FUNCTION_BLOCK UA_SkillFacade (* OPC UA object of one skill: one method per PackML command (answered synchronously with Accepted/ErrorID) and published State, ErrorID and latched parameters *)
  (* Standard: 61499-2 *)
  (* Version 2.0, 2026-09-27, Project contributors, Filling cell reference model *)
  PACKAGE fillingcell;
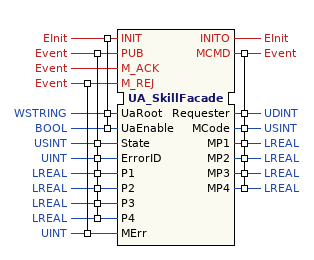
  EVENT_INPUT
    INIT : EInit WITH UaRoot, UaEnable;
    PUB WITH State, ErrorID, P1, P2, P3, P4;
    M_ACK;
    M_REJ WITH MErr;
  END_EVENT
  EVENT_OUTPUT
    INITO : EInit;
    MCMD WITH Requester, MCode, MP1, MP2, MP3, MP4;
  END_EVENT
  VAR_INPUT
    UaRoot : WSTRING;
    UaEnable : BOOL;
    State : USINT;
    ErrorID : UINT;
    P1 : LREAL;
    P2 : LREAL;
    P3 : LREAL;
    P4 : LREAL;
    MErr : UINT;
  END_VAR
  VAR_OUTPUT
    Requester : UDINT;
    MCode : USINT;
    MP1 : LREAL;
    MP2 : LREAL;
    MP3 : LREAL;
    MP4 : LREAL;
  END_VAR
  FBS
    Ids : fillingcell::UA_SkillIds;
    Calls : fillingcell::UA_SkillMux;
    Srv_Reset : iec61499::net::SERVER_2_1;
    Srv_Start : iec61499::net::SERVER_2_5;
    Srv_Hold : iec61499::net::SERVER_2_1;
    Srv_Unhold : iec61499::net::SERVER_2_1;
    Srv_Stop : iec61499::net::SERVER_2_1;
    Srv_Abort : iec61499::net::SERVER_2_1;
    Srv_Clear : iec61499::net::SERVER_2_1;
    Publisher : iec61499::net::PUBLISH_6;
  END_FBS
  EVENT_CONNECTIONS
    Srv_Reset.IND TO Calls.IND_Reset;
    Calls.RSP_Reset TO Srv_Reset.RSP;
    Srv_Start.IND TO Calls.IND_Start;
    Calls.RSP_Start TO Srv_Start.RSP;
    Srv_Hold.IND TO Calls.IND_Hold;
    Calls.RSP_Hold TO Srv_Hold.RSP;
    Srv_Unhold.IND TO Calls.IND_Unhold;
    Calls.RSP_Unhold TO Srv_Unhold.RSP;
    Srv_Stop.IND TO Calls.IND_Stop;
    Calls.RSP_Stop TO Srv_Stop.RSP;
    Srv_Abort.IND TO Calls.IND_Abort;
    Calls.RSP_Abort TO Srv_Abort.RSP;
    Srv_Clear.IND TO Calls.IND_Clear;
    Calls.RSP_Clear TO Srv_Clear.RSP;
    INIT TO Ids.INIT;
    Ids.INITO TO Srv_Reset.INIT;
    Srv_Reset.INITO TO Srv_Start.INIT;
    Srv_Start.INITO TO Srv_Hold.INIT;
    Srv_Hold.INITO TO Srv_Unhold.INIT;
    Srv_Unhold.INITO TO Srv_Stop.INIT;
    Srv_Stop.INITO TO Srv_Abort.INIT;
    Srv_Abort.INITO TO Srv_Clear.INIT;
    Srv_Clear.INITO TO Publisher.INIT;
    Publisher.INITO TO INITO;
    PUB TO Publisher.REQ;
    Calls.S_CMD TO MCMD;
    M_ACK TO Calls.S_ACK;
    M_REJ TO Calls.S_REJ;
  END_CONNECTIONS
  DATA_CONNECTIONS
    UaEnable TO Srv_Reset.QI;
    Ids.Id_Reset TO Srv_Reset.ID;
    Srv_Reset.RD_1 TO Calls.Req_Reset;
    Calls.Accepted TO Srv_Reset.SD_1;
    Calls.ErrorID TO Srv_Reset.SD_2;
    UaEnable TO Srv_Start.QI;
    Ids.Id_Start TO Srv_Start.ID;
    Srv_Start.RD_1 TO Calls.Req_Start;
    Srv_Start.RD_2 TO Calls.Start_P1;
    Srv_Start.RD_3 TO Calls.Start_P2;
    Srv_Start.RD_4 TO Calls.Start_P3;
    Srv_Start.RD_5 TO Calls.Start_P4;
    Calls.Accepted TO Srv_Start.SD_1;
    Calls.ErrorID TO Srv_Start.SD_2;
    UaEnable TO Srv_Hold.QI;
    Ids.Id_Hold TO Srv_Hold.ID;
    Srv_Hold.RD_1 TO Calls.Req_Hold;
    Calls.Accepted TO Srv_Hold.SD_1;
    Calls.ErrorID TO Srv_Hold.SD_2;
    UaEnable TO Srv_Unhold.QI;
    Ids.Id_Unhold TO Srv_Unhold.ID;
    Srv_Unhold.RD_1 TO Calls.Req_Unhold;
    Calls.Accepted TO Srv_Unhold.SD_1;
    Calls.ErrorID TO Srv_Unhold.SD_2;
    UaEnable TO Srv_Stop.QI;
    Ids.Id_Stop TO Srv_Stop.ID;
    Srv_Stop.RD_1 TO Calls.Req_Stop;
    Calls.Accepted TO Srv_Stop.SD_1;
    Calls.ErrorID TO Srv_Stop.SD_2;
    UaEnable TO Srv_Abort.QI;
    Ids.Id_Abort TO Srv_Abort.ID;
    Srv_Abort.RD_1 TO Calls.Req_Abort;
    Calls.Accepted TO Srv_Abort.SD_1;
    Calls.ErrorID TO Srv_Abort.SD_2;
    UaEnable TO Srv_Clear.QI;
    Ids.Id_Clear TO Srv_Clear.ID;
    Srv_Clear.RD_1 TO Calls.Req_Clear;
    Calls.Accepted TO Srv_Clear.SD_1;
    Calls.ErrorID TO Srv_Clear.SD_2;
    UaRoot TO Ids.UaRoot;
    UaEnable TO Publisher.QI;
    Ids.IdPub TO Publisher.ID;
    State TO Publisher.SD_1;
    ErrorID TO Publisher.SD_2;
    P1 TO Publisher.SD_3;
    P2 TO Publisher.SD_4;
    P3 TO Publisher.SD_5;
    P4 TO Publisher.SD_6;
    MErr TO Calls.S_Err;
    Calls.Requester TO Requester;
    Calls.S_Code TO MCode;
    Calls.S_P1 TO MP1;
    Calls.S_P2 TO MP2;
    Calls.S_P3 TO MP3;
    Calls.S_P4 TO MP4;
  END_CONNECTIONS
END_FUNCTION_BLOCK
